// TIA Portal V17 export
// export: Created 2024-09-02T12:50:00.9082389Z, ExportSetting WithDefaults, DisplayName Totally Integrated Automation Portal, DisplayVersion V17, DisplayName TIA Portal Openness, DisplayVersion V17, DisplayName TIA Portal Version Control Interface, DisplayVersion V17, DisplayName STEP 7 Professional, DisplayVersion V17, DisplayName STEP 7 Safety, DisplayVersion V17, DisplayName WinCC Professional, DisplayVersion V17
FUNCTION_BLOCK "GraFB_Hand_41_50"   // FB1174, GRAPH
TITLE = GRAPH FB
AUTHOR : OlegFuehrus
FAMILY : SK
NAME : SK
VERSION : 0.1
// Hand functions / Handfunktionen
// stored: AcknowledgeErrorsRequired true, AutoNumber true, ExtensionBlockName LTLL_ManualGraphExt, GraphVersion 4.0, InitialValuesAcquisition false, IsIECCheckEnabled false, LanguageInNetworks LAD, LockOperatingMode false, PermanentILProcessingInMANMode true, SetENOAutomatically false, SkipSteps false, UDAEnableTagReadback false, WithAlarmHandling true
   // inherited from GRAPH_BASE
   VAR
      OFF_SQ_BASE : Bool;
   END_VAR
   VAR_INPUT
      OFF_SQ : Bool;
      INIT_SQ : Bool;
      ACK_EF : Bool;
      S_PREV : Bool;
      S_NEXT : Bool;
      SW_AUTO : Bool;
      SW_TAP : Bool;
      SW_MAN : Bool;
      S_SEL : Int;
      S_ON : Bool;
      S_OFF : Bool;
      T_PUSH : Bool;
   END_VAR
   VAR_OUTPUT
      S_NO : Int;
      S_MORE : Bool;
      S_ACTIVE : Bool;
      ERR_FLT : Bool;
      AUTO_ON : Bool;
      TAP_ON : Bool;
      MAN_ON : Bool;
   END_VAR
   VAR
      extBlock { S7_SetPoint := 'True'} : "LTLL_ManualGraphExt";
   END_VAR
   VAR_TEMP
      t_FrgHand : Bool;   // Freigabe Handbetrieb / Enable manual operation
      t_Service : Bool;   // Servicebetrieb aktiv / Service operation active
   END_VAR
BEGIN
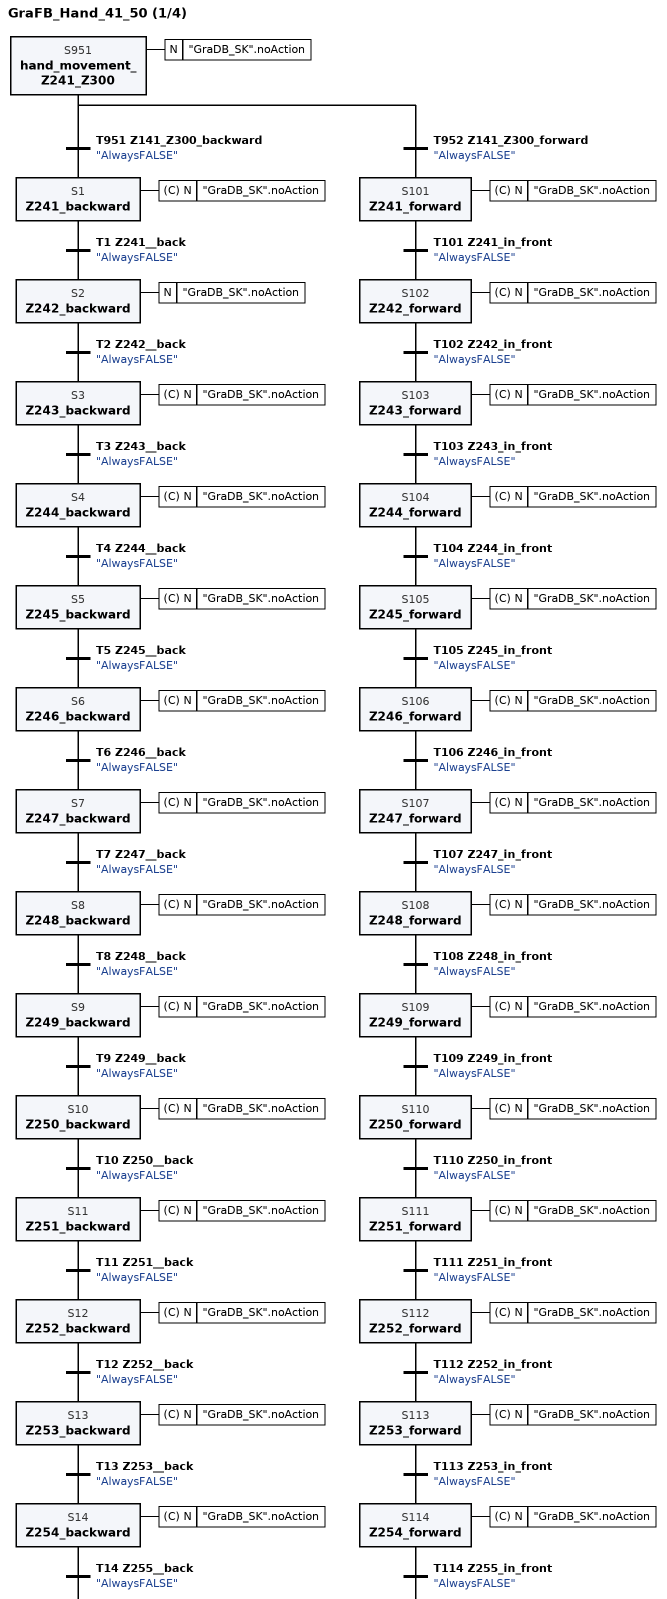
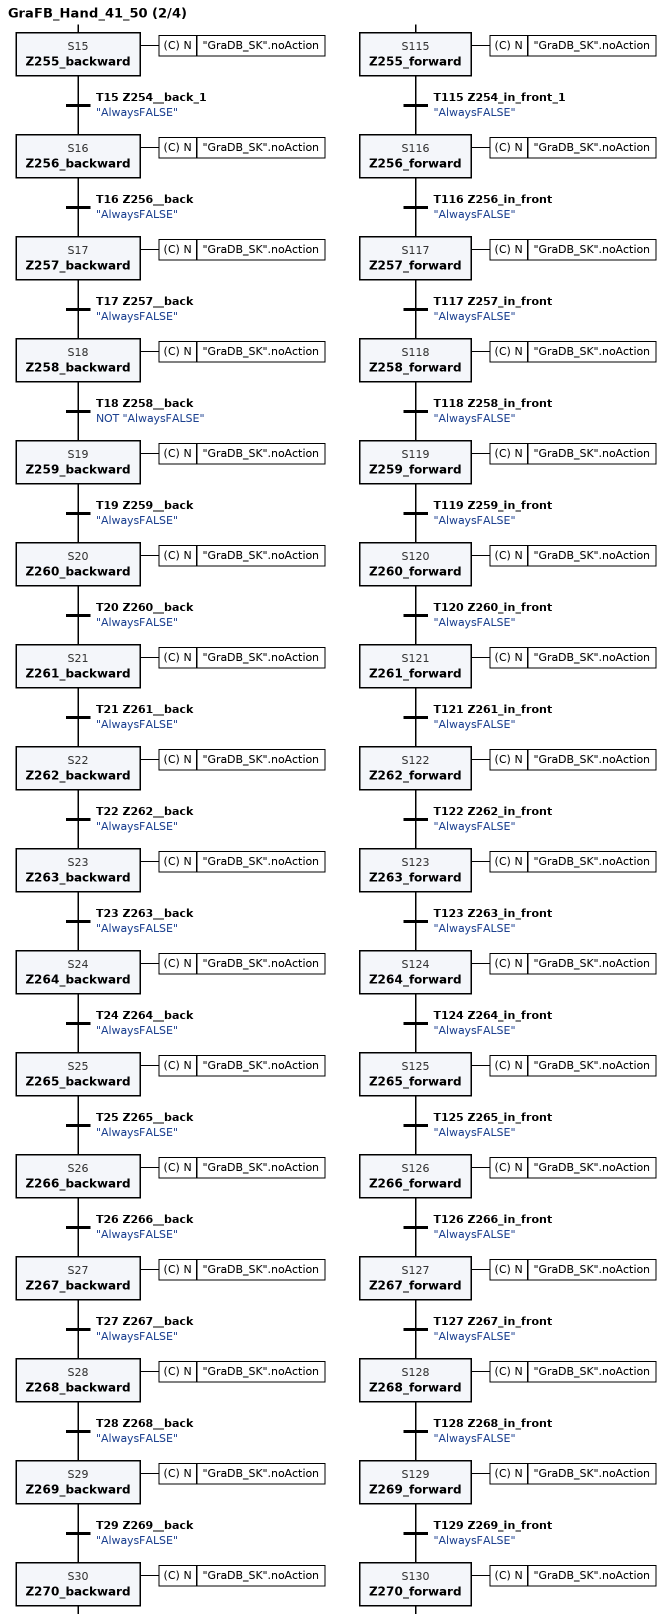
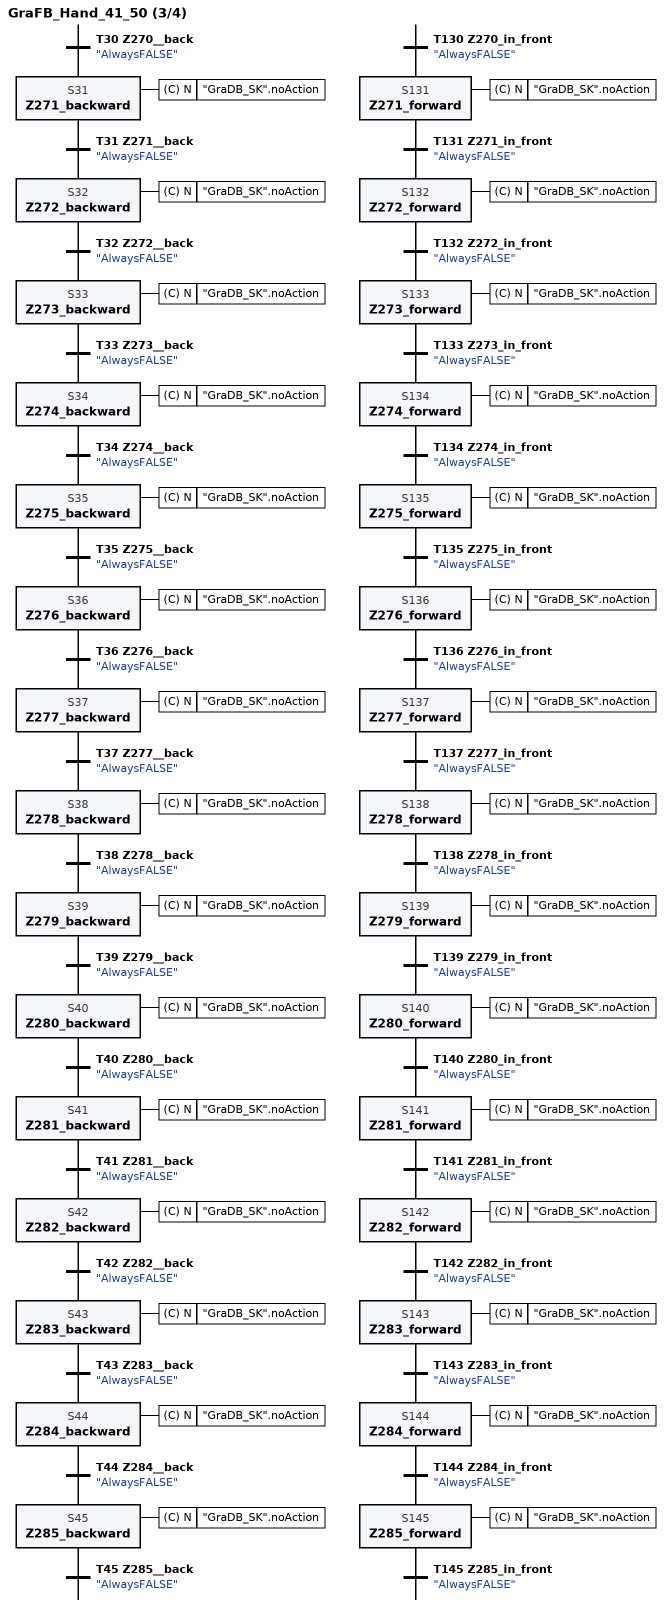
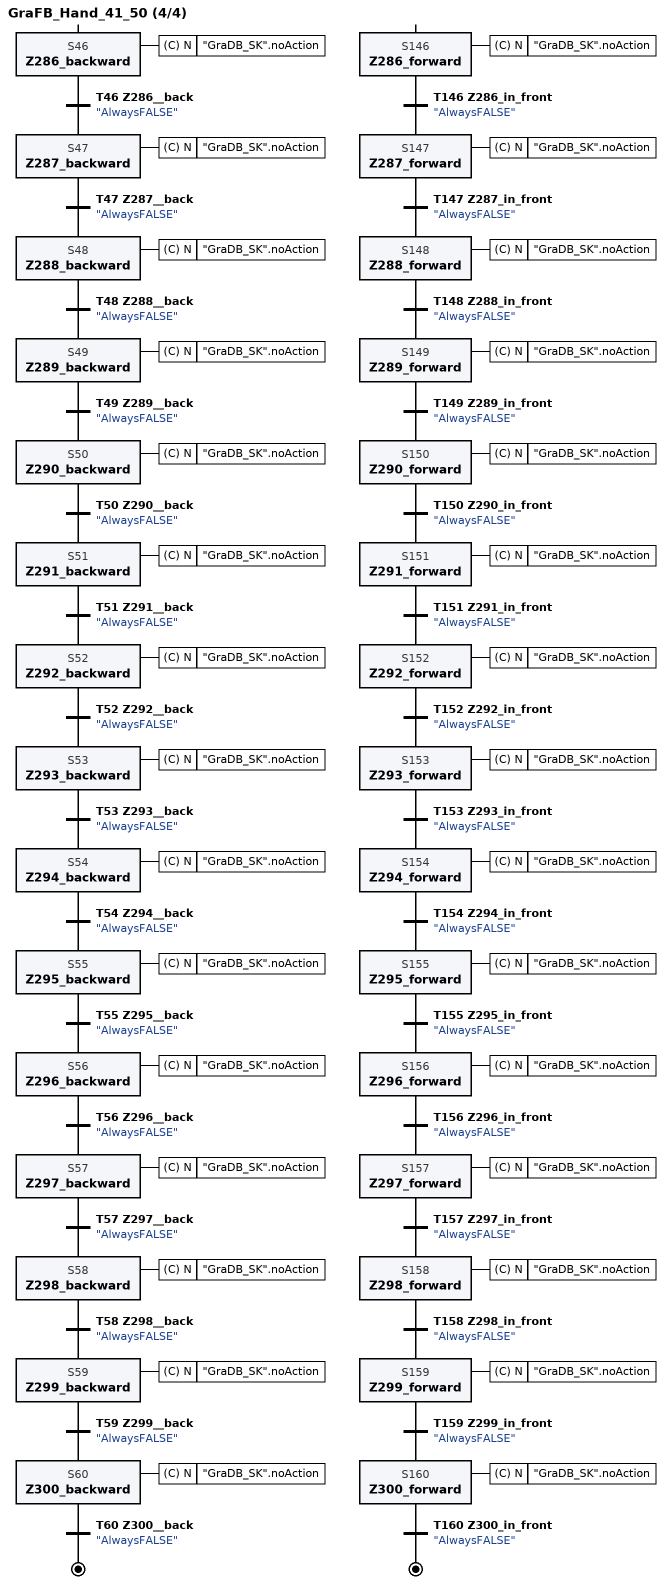
   // permanent pre-instructions
   NETWORK 1
   TITLE = HMI Lite Pass on data / HMI Lite Daten weiterreichen
      #extBlock.input := "LTLL_ManualGraphControl_OP70".screen[0].input;
   NETWORK 2
   TITLE = Instance DB Name query and pass on / Instanz DB Name abfragen und weiterreichen
      GetInstanceName(size := 0, OUT => #extBlock.input.instanceName);
   NETWORK 3
   TITLE = Interlocks Permanent machining, manual Approve and service / Interlocks Permanent Bearbeiten, Handfreigabe und Service
      IF NOT #RT_DATA.MOP.IL_PERM THEN #RT_DATA.MOP.IL_PERM := TRUE; END_IF;
      #t_FrgHand := "AnwDB_OperatingModes_OP70".BA[0]."mode_hand+start";
      #t_Service := "AnwDB_OperatingModes_OP70".BA[0].mode_service;

   // sequencer 1: Sequencer 1
   STEP hand_movement_Z241_Z300:   // S951, max time T#10S, warning time T#7S: Step commentary / Schrittkommentar
      interlock C := (none);   // hand_bereich_Z001_Z005
      supervision V := (none);   // hand_bereich_Z001_Z005
              N    "GraDB_SK".noAction
   END_STEP
   TRANSITION Z141_Z300_backward FROM hand_movement_Z241_Z300 TO Z241_backward   // T951
      := "AlwaysFALSE";
   END_TRANSITION
   TRANSITION Z141_Z300_forward FROM hand_movement_Z241_Z300 TO Z241_forward   // T952
      := "AlwaysFALSE";
   END_TRANSITION
   STEP Z241_backward:   // S1, max time T#10S, warning time T#7S
      interlock C := "AlwaysFALSE";   // Z241_zur
      supervision V := NOT #Z241__back.TT AND (#Z241_backward.T > T#5S);   // Z241_zur
      (C)     N    "GraDB_SK".noAction
   END_STEP
   TRANSITION Z241__back FROM Z241_backward TO Z242_backward   // T1
      := "AlwaysFALSE";
   END_TRANSITION
   STEP Z242_backward:   // S2, max time T#10S, warning time T#7S
      interlock C := "AlwaysFALSE";   // Z242_zur
      supervision V := NOT #Z242__back.TT AND (#Z242_backward.T > T#5S);   // Z242_zur
              N    "GraDB_SK".noAction
   END_STEP
   TRANSITION Z242__back FROM Z242_backward TO Z243_backward   // T2
      := "AlwaysFALSE";
   END_TRANSITION
   STEP Z243_backward:   // S3, max time T#10S, warning time T#7S
      interlock C := "AlwaysFALSE";   // Z243_zur
      supervision V := NOT #Z243__back.TT AND (#Z243_backward.T > T#5S);   // Z243_zur
      (C)     N    "GraDB_SK".noAction
   END_STEP
   TRANSITION Z243__back FROM Z243_backward TO Z244_backward   // T3
      := "AlwaysFALSE";
   END_TRANSITION
   STEP Z244_backward:   // S4, max time T#10S, warning time T#7S
      interlock C := "AlwaysFALSE";   // Z244_zur
      supervision V := NOT #Z244__back.TT AND (#Z244_backward.T > T#5S);   // Z244_zur
      (C)     N    "GraDB_SK".noAction
   END_STEP
   TRANSITION Z244__back FROM Z244_backward TO Z245_backward   // T4
      := "AlwaysFALSE";
   END_TRANSITION
   STEP Z245_backward:   // S5, max time T#10S, warning time T#7S
      interlock C := "AlwaysFALSE";   // Z245_zur
      supervision V := NOT #Z245__back.TT AND (#Z245_backward.T > T#5S);   // Z245_zur
      (C)     N    "GraDB_SK".noAction
   END_STEP
   TRANSITION Z245__back FROM Z245_backward TO Z246_backward   // T5
      := "AlwaysFALSE";
   END_TRANSITION
   STEP Z241_forward:   // S101, max time T#10S, warning time T#7S
      interlock C := "AlwaysFALSE";   // Z241_vor
      supervision V := NOT #Z241_in_front.TT AND (#Z241_forward.T > T#5S);   // Z241_vor
      (C)     N    "GraDB_SK".noAction
   END_STEP
   TRANSITION Z241_in_front FROM Z241_forward TO Z242_forward   // T101
      := "AlwaysFALSE";
   END_TRANSITION
   STEP Z242_forward:   // S102, max time T#10S, warning time T#7S
      interlock C := "AlwaysFALSE";   // Z242_vor
      supervision V := NOT #Z242_in_front.TT AND (#Z242_forward.T > T#5S);   // Z242_vor
      (C)     N    "GraDB_SK".noAction
   END_STEP
   TRANSITION Z242_in_front FROM Z242_forward TO Z243_forward   // T102
      := "AlwaysFALSE";
   END_TRANSITION
   STEP Z243_forward:   // S103, max time T#10S, warning time T#7S
      interlock C := "AlwaysFALSE";   // Z243_vor
      supervision V := NOT #Z243_in_front.TT AND (#Z243_forward.T > T#5S);   // Z243_vor
      (C)     N    "GraDB_SK".noAction
   END_STEP
   TRANSITION Z243_in_front FROM Z243_forward TO Z244_forward   // T103
      := "AlwaysFALSE";
   END_TRANSITION
   STEP Z244_forward:   // S104, max time T#10S, warning time T#7S
      interlock C := "AlwaysFALSE";   // Z244_vor
      supervision V := NOT #Z244_in_front.TT AND (#Z244_forward.T > T#5S);   // Z244_vor
      (C)     N    "GraDB_SK".noAction
   END_STEP
   TRANSITION Z244_in_front FROM Z244_forward TO Z245_forward   // T104
      := "AlwaysFALSE";
   END_TRANSITION
   STEP Z245_forward:   // S105, max time T#10S, warning time T#7S
      interlock C := "AlwaysFALSE";   // Z245_vor
      supervision V := NOT #Z245_in_front.TT AND (#Z245_forward.T > T#20S);   // Z245_vor
      (C)     N    "GraDB_SK".noAction
   END_STEP
   TRANSITION Z245_in_front FROM Z245_forward TO Z246_forward   // T105
      := "AlwaysFALSE";
   END_TRANSITION
   STEP Z246_backward:   // S6, max time T#10S, warning time T#7S: Cross transport 2 / Quertransport 2
      interlock C := "AlwaysFALSE";   // Z246_zur
      supervision V := NOT #Z246__back.TT AND (#Z246_backward.T > T#5S);   // Z246_zur
      (C)     N    "GraDB_SK".noAction
   END_STEP
   TRANSITION Z246__back FROM Z246_backward TO Z247_backward   // T6
      := "AlwaysFALSE";
   END_TRANSITION
   STEP Z247_backward:   // S7, max time T#10S, warning time T#7S
      interlock C := "AlwaysFALSE";   // Z247_zur
      supervision V := NOT #Z247__back.TT AND (#Z247_backward.T > T#5S);   // Z247_zur
      (C)     N    "GraDB_SK".noAction
   END_STEP
   TRANSITION Z247__back FROM Z247_backward TO Z248_backward   // T7
      := "AlwaysFALSE";
   END_TRANSITION
   STEP Z248_backward:   // S8, max time T#10S, warning time T#7S
      interlock C := "AlwaysFALSE";   // Z248_zur
      supervision V := NOT #Z248__back.TT AND (#Z248_backward.T > T#5S);   // Z248_zur
      (C)     N    "GraDB_SK".noAction
   END_STEP
   TRANSITION Z248__back FROM Z248_backward TO Z249_backward   // T8
      := "AlwaysFALSE";
   END_TRANSITION
   STEP Z249_backward:   // S9, max time T#10S, warning time T#7S
      interlock C := "AlwaysFALSE";   // Z249_zur
      supervision V := NOT #Z249__back.TT AND (#Z249_backward.T > T#5S);   // Z249_zur
      (C)     N    "GraDB_SK".noAction
   END_STEP
   TRANSITION Z249__back FROM Z249_backward TO Z250_backward   // T9
      := "AlwaysFALSE";
   END_TRANSITION
   STEP Z250_backward:   // S10, max time T#10S, warning time T#7S
      interlock C := "AlwaysFALSE";   // Z250_zur
      supervision V := NOT #Z250__back.TT AND (#Z250_backward.T > T#5S);   // Z250_zur
      (C)     N    "GraDB_SK".noAction
   END_STEP
   TRANSITION Z250__back FROM Z250_backward TO Z251_backward   // T10
      := "AlwaysFALSE";
   END_TRANSITION
   STEP Z246_forward:   // S106, max time T#10S, warning time T#7S
      interlock C := "AlwaysFALSE";   // Z246_vor
      supervision V := NOT #Z246_in_front.TT AND (#Z246_forward.T > T#5S);   // Z246_vor
      (C)     N    "GraDB_SK".noAction
   END_STEP
   TRANSITION Z246_in_front FROM Z246_forward TO Z247_forward   // T106
      := "AlwaysFALSE";
   END_TRANSITION
   STEP Z247_forward:   // S107, max time T#10S, warning time T#7S
      interlock C := "AlwaysFALSE";   // Z247_vor
      supervision V := NOT #Z247_in_front.TT AND (#Z247_forward.T > T#5S);   // Z247_vor
      (C)     N    "GraDB_SK".noAction
   END_STEP
   TRANSITION Z247_in_front FROM Z247_forward TO Z248_forward   // T107
      := "AlwaysFALSE";
   END_TRANSITION
   STEP Z248_forward:   // S108, max time T#10S, warning time T#7S
      interlock C := "AlwaysFALSE";   // Z248_vor
      supervision V := NOT #Z248_in_front.TT AND (#Z248_forward.T > T#5S);   // Z248_vor
      (C)     N    "GraDB_SK".noAction
   END_STEP
   TRANSITION Z248_in_front FROM Z248_forward TO Z249_forward   // T108
      := "AlwaysFALSE";
   END_TRANSITION
   STEP Z249_forward:   // S109, max time T#10S, warning time T#7S
      interlock C := "AlwaysFALSE";   // Z249_vor
      supervision V := NOT #Z249_in_front.TT AND (#Z249_forward.T > T#5S);   // Z249_vor
      (C)     N    "GraDB_SK".noAction
   END_STEP
   TRANSITION Z249_in_front FROM Z249_forward TO Z250_forward   // T109
      := "AlwaysFALSE";
   END_TRANSITION
   STEP Z250_forward:   // S110, max time T#10S, warning time T#7S
      interlock C := "AlwaysFALSE";   // Z250_vor
      supervision V := NOT #Z250_in_front.TT AND (#Z250_forward.T > T#5S);   // Z250_vor
      (C)     N    "GraDB_SK".noAction
   END_STEP
   TRANSITION Z250_in_front FROM Z250_forward TO Z251_forward   // T110
      := "AlwaysFALSE";
   END_TRANSITION
   STEP Z251_backward:   // S11, max time T#10S, warning time T#7S
      interlock C := "AlwaysFALSE";   // Z251_zur
      supervision V := NOT #Z251__back.TT AND (#Z251_backward.T > T#5S);   // Z251_zur
      (C)     N    "GraDB_SK".noAction
   END_STEP
   TRANSITION Z251__back FROM Z251_backward TO Z252_backward   // T11
      := "AlwaysFALSE";
   END_TRANSITION
   STEP Z252_backward:   // S12, max time T#10S, warning time T#7S
      interlock C := "AlwaysFALSE";   // Z252_zur
      supervision V := NOT #Z252__back.TT AND (#Z252_backward.T > T#5S);   // Z252_zur
      (C)     N    "GraDB_SK".noAction
   END_STEP
   TRANSITION Z252__back FROM Z252_backward TO Z253_backward   // T12
      := "AlwaysFALSE";
   END_TRANSITION
   STEP Z253_backward:   // S13, max time T#10S, warning time T#7S
      interlock C := "AlwaysFALSE";   // Z253_zur
      supervision V := NOT #Z253__back.TT AND (#Z253_backward.T > T#5S);   // Z253_zur
      (C)     N    "GraDB_SK".noAction
   END_STEP
   TRANSITION Z253__back FROM Z253_backward TO Z254_backward   // T13
      := "AlwaysFALSE";
   END_TRANSITION
   STEP Z254_backward:   // S14, max time T#10S, warning time T#7S
      interlock C := "AlwaysFALSE";   // Z255_zur
      supervision V := NOT #Z255__back.TT AND (#Z254_backward.T > T#5S);   // Z255_zur
      (C)     N    "GraDB_SK".noAction
   END_STEP
   TRANSITION Z255__back FROM Z254_backward TO Z255_backward   // T14
      := "AlwaysFALSE";
   END_TRANSITION
   STEP Z255_backward:   // S15, max time T#10S, warning time T#7S
      interlock C := "AlwaysFALSE";   // Z254_zur
      supervision V := NOT #Z256__back.TT AND (#Z255_backward.T > T#5S);   // Z25_zur
      (C)     N    "GraDB_SK".noAction
   END_STEP
   TRANSITION Z254__back_1 FROM Z255_backward TO Z256_backward   // T15
      := "AlwaysFALSE";
   END_TRANSITION
   STEP Z251_forward:   // S111, max time T#10S, warning time T#7S
      interlock C := "AlwaysFALSE";   // Z251_vor
      supervision V := NOT #Z251_in_front.TT AND (#Z251_forward.T > T#5S);   // Z251_vor
      (C)     N    "GraDB_SK".noAction
   END_STEP
   TRANSITION Z251_in_front FROM Z251_forward TO Z252_forward   // T111
      := "AlwaysFALSE";
   END_TRANSITION
   STEP Z252_forward:   // S112, max time T#10S, warning time T#7S
      interlock C := "AlwaysFALSE";   // Z252_vor
      supervision V := NOT #Z252_in_front.TT AND (#Z252_forward.T > T#5S);   // Z252_vor
      (C)     N    "GraDB_SK".noAction
   END_STEP
   TRANSITION Z252_in_front FROM Z252_forward TO Z253_forward   // T112
      := "AlwaysFALSE";
   END_TRANSITION
   STEP Z253_forward:   // S113, max time T#10S, warning time T#7S
      interlock C := "AlwaysFALSE";   // Z253_vor
      supervision V := NOT #Z253_in_front.TT AND (#Z253_forward.T > T#5S);   // Z253_vor
      (C)     N    "GraDB_SK".noAction
   END_STEP
   TRANSITION Z253_in_front FROM Z253_forward TO Z254_forward   // T113
      := "AlwaysFALSE";
   END_TRANSITION
   STEP Z254_forward:   // S114, max time T#10S, warning time T#7S
      interlock C := "AlwaysFALSE";   // Z255_vor
      supervision V := NOT #Z255_in_front.TT AND (#Z254_forward.T > T#5S);   // Z255_vor
      (C)     N    "GraDB_SK".noAction
   END_STEP
   TRANSITION Z255_in_front FROM Z254_forward TO Z255_forward   // T114
      := "AlwaysFALSE";
   END_TRANSITION
   STEP Z255_forward:   // S115, max time T#10S, warning time T#7S
      interlock C := "AlwaysFALSE";   // Z254_vor
      supervision V := NOT #Z256_in_front.TT AND (#Z255_forward.T > T#5S);   // Z254_vor
      (C)     N    "GraDB_SK".noAction
   END_STEP
   TRANSITION Z254_in_front_1 FROM Z255_forward TO Z256_forward   // T115
      := "AlwaysFALSE";
   END_TRANSITION
   STEP Z256_backward:   // S16, max time T#10S, warning time T#7S
      interlock C := "AlwaysFALSE";   // Z256_zur
      supervision V := NOT #Z256__back.TT AND (#Z256_backward.T > T#5S);   // Z256_zur
      (C)     N    "GraDB_SK".noAction
   END_STEP
   TRANSITION Z256__back FROM Z256_backward TO Z257_backward   // T16
      := "AlwaysFALSE";
   END_TRANSITION
   STEP Z257_backward:   // S17, max time T#10S, warning time T#7S
      interlock C := "AlwaysFALSE";   // Z257_zur
      supervision V := NOT #Z257__back.TT AND (#Z257_backward.T > T#5S);   // Z257_zur
      (C)     N    "GraDB_SK".noAction
   END_STEP
   TRANSITION Z257__back FROM Z257_backward TO Z258_backward   // T17
      := "AlwaysFALSE";
   END_TRANSITION
   STEP Z258_backward:   // S18, max time T#10S, warning time T#7S
      interlock C := "AlwaysFALSE";   // Z258_zur
      supervision V := NOT #Z258__back.TT AND (#Z258_backward.T > T#5S);   // Z258_zur
      (C)     N    "GraDB_SK".noAction
   END_STEP
   TRANSITION Z258__back FROM Z258_backward TO Z259_backward   // T18
      := NOT "AlwaysFALSE";
   END_TRANSITION
   STEP Z259_backward:   // S19, max time T#10S, warning time T#7S
      interlock C := "AlwaysFALSE";   // Z259_zur
      supervision V := NOT #Z259__back.TT AND (#Z259_backward.T > T#5S);   // Z259_zur
      (C)     N    "GraDB_SK".noAction
   END_STEP
   TRANSITION Z259__back FROM Z259_backward TO Z260_backward   // T19
      := "AlwaysFALSE";
   END_TRANSITION
   STEP Z260_backward:   // S20, max time T#10S, warning time T#7S
      interlock C := "AlwaysFALSE";   // Z260_zur
      supervision V := NOT #Z260__back.TT AND (#Z260_backward.T > T#5S);   // Z260_zur
      (C)     N    "GraDB_SK".noAction
   END_STEP
   TRANSITION Z260__back FROM Z260_backward TO Z261_backward   // T20
      := "AlwaysFALSE";
   END_TRANSITION
   STEP Z256_forward:   // S116, max time T#10S, warning time T#7S
      interlock C := "AlwaysFALSE";   // Z256_vor
      supervision V := NOT #Z256_in_front.TT AND (#Z256_forward.T > T#5S);   // Z256_vor
      (C)     N    "GraDB_SK".noAction
   END_STEP
   TRANSITION Z256_in_front FROM Z256_forward TO Z257_forward   // T116
      := "AlwaysFALSE";
   END_TRANSITION
   STEP Z257_forward:   // S117, max time T#10S, warning time T#7S
      interlock C := "AlwaysFALSE";   // Z257_vor
      supervision V := NOT #Z257_in_front.TT AND (#Z257_forward.T > T#5S);   // Z257_vor
      (C)     N    "GraDB_SK".noAction
   END_STEP
   TRANSITION Z257_in_front FROM Z257_forward TO Z258_forward   // T117
      := "AlwaysFALSE";
   END_TRANSITION
   STEP Z258_forward:   // S118, max time T#10S, warning time T#7S
      interlock C := "AlwaysFALSE";   // Z258_vor
      supervision V := NOT #Z258_in_front.TT AND (#Z258_forward.T > T#5S);   // Z258_vor
      (C)     N    "GraDB_SK".noAction
   END_STEP
   TRANSITION Z258_in_front FROM Z258_forward TO Z259_forward   // T118
      := "AlwaysFALSE";
   END_TRANSITION
   STEP Z259_forward:   // S119, max time T#10S, warning time T#7S
      interlock C := "AlwaysFALSE";   // Z259_vor
      supervision V := NOT #Z259_in_front.TT AND (#Z259_forward.T > T#5S);   // Z259_vor
      (C)     N    "GraDB_SK".noAction
   END_STEP
   TRANSITION Z259_in_front FROM Z259_forward TO Z260_forward   // T119
      := "AlwaysFALSE";
   END_TRANSITION
   STEP Z260_forward:   // S120, max time T#10S, warning time T#7S
      interlock C := "AlwaysFALSE";   // Z260_vor
      supervision V := NOT #Z260_in_front.TT AND (#Z260_forward.T > T#5S);   // Z260_vor
      (C)     N    "GraDB_SK".noAction
   END_STEP
   TRANSITION Z260_in_front FROM Z260_forward TO Z261_forward   // T120
      := "AlwaysFALSE";
   END_TRANSITION
   STEP Z261_backward:   // S21, max time T#10S, warning time T#7S
      interlock C := "AlwaysFALSE";   // Z261_zur
      supervision V := NOT #Z261__back.TT AND (#Z261_backward.T > T#10S);   // Z261_zur
      (C)     N    "GraDB_SK".noAction
   END_STEP
   TRANSITION Z261__back FROM Z261_backward TO Z262_backward   // T21
      := "AlwaysFALSE";
   END_TRANSITION
   STEP Z262_backward:   // S22, max time T#10S, warning time T#7S
      interlock C := "AlwaysFALSE";   // Z262_zur
      supervision V := NOT #Z262__back.TT AND (#Z262_backward.T > T#10S);   // Z262_zur
      (C)     N    "GraDB_SK".noAction
   END_STEP
   TRANSITION Z262__back FROM Z262_backward TO Z263_backward   // T22
      := "AlwaysFALSE";
   END_TRANSITION
   STEP Z263_backward:   // S23, max time T#10S, warning time T#7S
      interlock C := "AlwaysFALSE";   // Z263_zur
      supervision V := NOT #Z263__back.TT AND (#Z263_backward.T > T#10S);   // Z263_zur
      (C)     N    "GraDB_SK".noAction
   END_STEP
   TRANSITION Z263__back FROM Z263_backward TO Z264_backward   // T23
      := "AlwaysFALSE";
   END_TRANSITION
   STEP Z264_backward:   // S24, max time T#10S, warning time T#7S
      interlock C := "AlwaysFALSE";   // Z264_zur
      supervision V := NOT #Z264__back.TT AND (#Z264_backward.T > T#5S);   // Z264_zur
      (C)     N    "GraDB_SK".noAction
   END_STEP
   TRANSITION Z264__back FROM Z264_backward TO Z265_backward   // T24
      := "AlwaysFALSE";
   END_TRANSITION
   STEP Z265_backward:   // S25, max time T#10S, warning time T#7S
      interlock C := "AlwaysFALSE";   // Z265_zur
      supervision V := NOT #Z265__back.TT AND (#Z265_backward.T > T#5S);   // Z265_zur
      (C)     N    "GraDB_SK".noAction
   END_STEP
   TRANSITION Z265__back FROM Z265_backward TO Z266_backward   // T25
      := "AlwaysFALSE";
   END_TRANSITION
   STEP Z261_forward:   // S121, max time T#10S, warning time T#7S
      interlock C := "AlwaysFALSE";   // Z261_vor
      supervision V := NOT #Z261_in_front.TT AND (#Z261_forward.T > T#5S);   // Z261_vor
      (C)     N    "GraDB_SK".noAction
   END_STEP
   TRANSITION Z261_in_front FROM Z261_forward TO Z262_forward   // T121
      := "AlwaysFALSE";
   END_TRANSITION
   STEP Z262_forward:   // S122, max time T#10S, warning time T#7S
      interlock C := "AlwaysFALSE";   // Z262_vor
      supervision V := NOT #Z262_in_front.TT AND (#Z262_forward.T > T#10S);   // Z262_vor
      (C)     N    "GraDB_SK".noAction
   END_STEP
   TRANSITION Z262_in_front FROM Z262_forward TO Z263_forward   // T122
      := "AlwaysFALSE";
   END_TRANSITION
   STEP Z263_forward:   // S123, max time T#10S, warning time T#7S
      interlock C := "AlwaysFALSE";   // Z263_vor
      supervision V := NOT #Z263_in_front.TT AND (#Z263_forward.T > T#10S);   // Z263_vor
      (C)     N    "GraDB_SK".noAction
   END_STEP
   TRANSITION Z263_in_front FROM Z263_forward TO Z264_forward   // T123
      := "AlwaysFALSE";
   END_TRANSITION
   STEP Z264_forward:   // S124, max time T#10S, warning time T#7S
      interlock C := "AlwaysFALSE";   // Z264_vor
      supervision V := NOT #Z264_in_front.TT AND (#Z264_forward.T > T#5S);   // Z264_vor
      (C)     N    "GraDB_SK".noAction
   END_STEP
   TRANSITION Z264_in_front FROM Z264_forward TO Z265_forward   // T124
      := "AlwaysFALSE";
   END_TRANSITION
   STEP Z265_forward:   // S125, max time T#10S, warning time T#7S
      interlock C := "AlwaysFALSE";   // Z265_vor
      supervision V := NOT #Z265_in_front.TT AND (#Z265_forward.T > T#5S);   // Z265_vor
      (C)     N    "GraDB_SK".noAction
   END_STEP
   TRANSITION Z265_in_front FROM Z265_forward TO Z266_forward   // T125
      := "AlwaysFALSE";
   END_TRANSITION
   STEP Z266_backward:   // S26, max time T#10S, warning time T#7S
      interlock C := "AlwaysFALSE";   // Z266_zur
      supervision V := NOT #Z266__back.TT AND (#Z266_backward.T > T#5S);   // Z266_zur
      (C)     N    "GraDB_SK".noAction
   END_STEP
   TRANSITION Z266__back FROM Z266_backward TO Z267_backward   // T26
      := "AlwaysFALSE";
   END_TRANSITION
   STEP Z267_backward:   // S27, max time T#10S, warning time T#7S
      interlock C := "AlwaysFALSE";   // Z267_zur
      supervision V := NOT #Z267__back.TT AND (#Z267_backward.T > T#5S);   // Z267_zur
      (C)     N    "GraDB_SK".noAction
   END_STEP
   TRANSITION Z267__back FROM Z267_backward TO Z268_backward   // T27
      := "AlwaysFALSE";
   END_TRANSITION
   STEP Z268_backward:   // S28, max time T#10S, warning time T#7S
      interlock C := "AlwaysFALSE";   // Z268_zur
      supervision V := NOT #Z268__back.TT AND (#Z268_backward.T > T#5S);   // Z268_zur
      (C)     N    "GraDB_SK".noAction
   END_STEP
   TRANSITION Z268__back FROM Z268_backward TO Z269_backward   // T28
      := "AlwaysFALSE";
   END_TRANSITION
   STEP Z269_backward:   // S29, max time T#10S, warning time T#7S
      interlock C := "AlwaysFALSE";   // Z269_zur
      supervision V := NOT #Z269__back.TT AND (#Z269_backward.T > T#5S);   // Z269_zur
      (C)     N    "GraDB_SK".noAction
   END_STEP
   TRANSITION Z269__back FROM Z269_backward TO Z270_backward   // T29
      := "AlwaysFALSE";
   END_TRANSITION
   STEP Z270_backward:   // S30, max time T#10S, warning time T#7S
      interlock C := "AlwaysFALSE";   // Z270_zur
      supervision V := NOT #Z270__back.TT AND (#Z270_backward.T > T#5S);   // Z270_zur
      (C)     N    "GraDB_SK".noAction
   END_STEP
   TRANSITION Z270__back FROM Z270_backward TO Z271_backward   // T30
      := "AlwaysFALSE";
   END_TRANSITION
   STEP Z266_forward:   // S126, max time T#10S, warning time T#7S
      interlock C := "AlwaysFALSE";   // Z266_vor
      supervision V := NOT #Z266_in_front.TT AND (#Z266_forward.T > T#5S);   // Z266_vor
      (C)     N    "GraDB_SK".noAction
   END_STEP
   TRANSITION Z266_in_front FROM Z266_forward TO Z267_forward   // T126
      := "AlwaysFALSE";
   END_TRANSITION
   STEP Z267_forward:   // S127, max time T#10S, warning time T#7S
      interlock C := "AlwaysFALSE";   // Z267_vor
      supervision V := NOT #Z267_in_front.TT AND (#Z267_forward.T > T#5S);   // Z267_vor
      (C)     N    "GraDB_SK".noAction
   END_STEP
   TRANSITION Z267_in_front FROM Z267_forward TO Z268_forward   // T127
      := "AlwaysFALSE";
   END_TRANSITION
   STEP Z268_forward:   // S128, max time T#10S, warning time T#7S
      interlock C := "AlwaysFALSE";   // Z268_vor
      supervision V := NOT #Z268_in_front.TT AND (#Z268_forward.T > T#5S);   // Z268_vor
      (C)     N    "GraDB_SK".noAction
   END_STEP
   TRANSITION Z268_in_front FROM Z268_forward TO Z269_forward   // T128
      := "AlwaysFALSE";
   END_TRANSITION
   STEP Z269_forward:   // S129, max time T#10S, warning time T#7S
      interlock C := "AlwaysFALSE";   // Z269_vor
      supervision V := NOT #Z269_in_front.TT AND (#Z269_forward.T > T#5S);   // Z269_vor
      (C)     N    "GraDB_SK".noAction
   END_STEP
   TRANSITION Z269_in_front FROM Z269_forward TO Z270_forward   // T129
      := "AlwaysFALSE";
   END_TRANSITION
   STEP Z270_forward:   // S130, max time T#10S, warning time T#7S
      interlock C := "AlwaysFALSE";   // Z270_vor
      supervision V := NOT #Z270_in_front.TT AND (#Z270_forward.T > T#5S);   // Z270_vor
      (C)     N    "GraDB_SK".noAction
   END_STEP
   TRANSITION Z270_in_front FROM Z270_forward TO Z271_forward   // T130
      := "AlwaysFALSE";
   END_TRANSITION
   STEP Z271_backward:   // S31, max time T#10S, warning time T#7S: Step commentary / Schrittkommentar
      interlock C := "AlwaysFALSE";   // Z271_zur
      supervision V := NOT #Z271__back.TT AND (#Z271_backward.T > T#5S);   // Z271_zur
      (C)     N    "GraDB_SK".noAction
   END_STEP
   TRANSITION Z271__back FROM Z271_backward TO Z272_backward   // T31
      := "AlwaysFALSE";
   END_TRANSITION
   STEP Z272_backward:   // S32, max time T#10S, warning time T#7S: Step commentary / Schrittkommentar
      interlock C := "AlwaysFALSE";   // Z272_zur
      supervision V := NOT #Z272__back.TT AND (#Z272_backward.T > T#5S);   // Z272_zur
      (C)     N    "GraDB_SK".noAction
   END_STEP
   TRANSITION Z272__back FROM Z272_backward TO Z273_backward   // T32
      := "AlwaysFALSE";
   END_TRANSITION
   STEP Z273_backward:   // S33, max time T#10S, warning time T#7S: Step commentary / Schrittkommentar
      interlock C := "AlwaysFALSE";   // Z273_zur
      supervision V := NOT #Z273__back.TT AND (#Z273_backward.T > T#5S);   // Z273_zur
      (C)     N    "GraDB_SK".noAction
   END_STEP
   TRANSITION Z273__back FROM Z273_backward TO Z274_backward   // T33
      := "AlwaysFALSE";
   END_TRANSITION
   STEP Z274_backward:   // S34, max time T#10S, warning time T#7S: Step commentary / Schrittkommentar
      interlock C := "AlwaysFALSE";   // Z274_zur
      supervision V := NOT #Z274__back.TT AND (#Z274_backward.T > T#5S);   // Z274_zur
      (C)     N    "GraDB_SK".noAction
   END_STEP
   TRANSITION Z274__back FROM Z274_backward TO Z275_backward   // T34
      := "AlwaysFALSE";
   END_TRANSITION
   STEP Z275_backward:   // S35, max time T#10S, warning time T#7S: Step commentary / Schrittkommentar
      interlock C := "AlwaysFALSE";   // Z275_zur
      supervision V := NOT #Z275__back.TT AND (#Z275_backward.T > T#5S);   // Z275_zur
      (C)     N    "GraDB_SK".noAction
   END_STEP
   TRANSITION Z275__back FROM Z275_backward TO Z276_backward   // T35
      := "AlwaysFALSE";
   END_TRANSITION
   STEP Z271_forward:   // S131, max time T#10S, warning time T#7S: Step commentary / Schrittkommentar
      interlock C := "AlwaysFALSE";   // Z271_vor
      supervision V := NOT #Z271_in_front.TT AND (#Z271_forward.T > T#5S);   // Z271_vor
      (C)     N    "GraDB_SK".noAction
   END_STEP
   TRANSITION Z271_in_front FROM Z271_forward TO Z272_forward   // T131
      := "AlwaysFALSE";
   END_TRANSITION
   STEP Z272_forward:   // S132, max time T#10S, warning time T#7S: Step commentary / Schrittkommentar
      interlock C := "AlwaysFALSE";   // Z272_vor
      supervision V := NOT #Z272_in_front.TT AND (#Z272_forward.T > T#5S);   // Z272_vor
      (C)     N    "GraDB_SK".noAction
   END_STEP
   TRANSITION Z272_in_front FROM Z272_forward TO Z273_forward   // T132
      := "AlwaysFALSE";
   END_TRANSITION
   STEP Z273_forward:   // S133, max time T#10S, warning time T#7S: Step commentary / Schrittkommentar
      interlock C := "AlwaysFALSE";   // Z273_vor
      supervision V := NOT #Z273_in_front.TT AND (#Z273_forward.T > T#5S);   // Z273_vor
      (C)     N    "GraDB_SK".noAction
   END_STEP
   TRANSITION Z273_in_front FROM Z273_forward TO Z274_forward   // T133
      := "AlwaysFALSE";
   END_TRANSITION
   STEP Z274_forward:   // S134, max time T#10S, warning time T#7S: Step commentary / Schrittkommentar
      interlock C := "AlwaysFALSE";   // Z274_vor
      supervision V := NOT #Z274_in_front.TT AND (#Z274_forward.T > T#5S);   // Z274_vor
      (C)     N    "GraDB_SK".noAction
   END_STEP
   TRANSITION Z274_in_front FROM Z274_forward TO Z275_forward   // T134
      := "AlwaysFALSE";
   END_TRANSITION
   STEP Z275_forward:   // S135, max time T#10S, warning time T#7S: Step commentary / Schrittkommentar
      interlock C := "AlwaysFALSE";   // Z275_vor
      supervision V := NOT #Z275_in_front.TT AND (#Z275_forward.T > T#5S);   // Z275_vor
      (C)     N    "GraDB_SK".noAction
   END_STEP
   TRANSITION Z275_in_front FROM Z275_forward TO Z276_forward   // T135
      := "AlwaysFALSE";
   END_TRANSITION
   STEP Z276_backward:   // S36, max time T#10S, warning time T#7S: Step commentary / Schrittkommentar
      interlock C := "AlwaysFALSE";   // Z276_zur
      supervision V := NOT #Z276__back.TT AND (#Z276_backward.T > T#5S);   // Z276_zur
      (C)     N    "GraDB_SK".noAction
   END_STEP
   TRANSITION Z276__back FROM Z276_backward TO Z277_backward   // T36
      := "AlwaysFALSE";
   END_TRANSITION
   STEP Z277_backward:   // S37, max time T#10S, warning time T#7S: Step commentary / Schrittkommentar
      interlock C := "AlwaysFALSE";   // Z277_zur
      supervision V := NOT #Z277__back.TT AND (#Z277_backward.T > T#5S);   // Z277_zur
      (C)     N    "GraDB_SK".noAction
   END_STEP
   TRANSITION Z277__back FROM Z277_backward TO Z278_backward   // T37
      := "AlwaysFALSE";
   END_TRANSITION
   STEP Z278_backward:   // S38, max time T#10S, warning time T#7S: Step commentary / Schrittkommentar
      interlock C := "AlwaysFALSE";   // Z278_zur
      supervision V := NOT #Z278__back.TT AND (#Z278_backward.T > T#5S);   // Z278_zur
      (C)     N    "GraDB_SK".noAction
   END_STEP
   TRANSITION Z278__back FROM Z278_backward TO Z279_backward   // T38
      := "AlwaysFALSE";
   END_TRANSITION
   STEP Z279_backward:   // S39, max time T#10S, warning time T#7S: Step commentary / Schrittkommentar
      interlock C := "AlwaysFALSE";   // Z279_zur
      supervision V := NOT #Z279__back.TT AND (#Z279_backward.T > T#5S);   // Z279_zur
      (C)     N    "GraDB_SK".noAction
   END_STEP
   TRANSITION Z279__back FROM Z279_backward TO Z280_backward   // T39
      := "AlwaysFALSE";
   END_TRANSITION
   STEP Z280_backward:   // S40, max time T#10S, warning time T#7S: Step commentary / Schrittkommentar
      interlock C := "AlwaysFALSE";   // Z280_zur
      supervision V := NOT #Z280__back.TT AND (#Z280_backward.T > T#5S);   // Z280_zur
      (C)     N    "GraDB_SK".noAction
   END_STEP
   TRANSITION Z280__back FROM Z280_backward TO Z281_backward   // T40
      := "AlwaysFALSE";
   END_TRANSITION
   STEP Z276_forward:   // S136, max time T#10S, warning time T#7S: Step commentary / Schrittkommentar
      interlock C := "AlwaysFALSE";   // Z276_vor
      supervision V := NOT #Z276_in_front.TT AND (#Z276_forward.T > T#5S);   // Z276_vor
      (C)     N    "GraDB_SK".noAction
   END_STEP
   TRANSITION Z276_in_front FROM Z276_forward TO Z277_forward   // T136
      := "AlwaysFALSE";
   END_TRANSITION
   STEP Z277_forward:   // S137, max time T#10S, warning time T#7S: Step commentary / Schrittkommentar
      interlock C := "AlwaysFALSE";   // Z277_vor
      supervision V := NOT #Z277_in_front.TT AND (#Z277_forward.T > T#5S);   // Z277_vor
      (C)     N    "GraDB_SK".noAction
   END_STEP
   TRANSITION Z277_in_front FROM Z277_forward TO Z278_forward   // T137
      := "AlwaysFALSE";
   END_TRANSITION
   STEP Z278_forward:   // S138, max time T#10S, warning time T#7S: Step commentary / Schrittkommentar
      interlock C := "AlwaysFALSE";   // Z278_vor
      supervision V := NOT #Z278_in_front.TT AND (#Z278_forward.T > T#5S);   // Z278_vor
      (C)     N    "GraDB_SK".noAction
   END_STEP
   TRANSITION Z278_in_front FROM Z278_forward TO Z279_forward   // T138
      := "AlwaysFALSE";
   END_TRANSITION
   STEP Z279_forward:   // S139, max time T#10S, warning time T#7S: Step commentary / Schrittkommentar
      interlock C := "AlwaysFALSE";   // Z279_vor
      supervision V := NOT #Z279_in_front.TT AND (#Z279_forward.T > T#5S);   // Z279_vor
      (C)     N    "GraDB_SK".noAction
   END_STEP
   TRANSITION Z279_in_front FROM Z279_forward TO Z280_forward   // T139
      := "AlwaysFALSE";
   END_TRANSITION
   STEP Z280_forward:   // S140, max time T#10S, warning time T#7S: Step commentary / Schrittkommentar
      interlock C := "AlwaysFALSE";   // Z280_vor
      supervision V := NOT #Z280_in_front.TT AND (#Z280_forward.T > T#5S);   // Z280_vor
      (C)     N    "GraDB_SK".noAction
   END_STEP
   TRANSITION Z280_in_front FROM Z280_forward TO Z281_forward   // T140
      := "AlwaysFALSE";
   END_TRANSITION
   STEP Z281_backward:   // S41, max time T#10S, warning time T#7S: Step commentary / Schrittkommentar
      interlock C := "AlwaysFALSE";   // Z281_zur
      supervision V := NOT #Z281__back.TT AND (#Z281_backward.T > T#5S);   // Z281_zur
      (C)     N    "GraDB_SK".noAction
   END_STEP
   TRANSITION Z281__back FROM Z281_backward TO Z282_backward   // T41
      := "AlwaysFALSE";
   END_TRANSITION
   STEP Z282_backward:   // S42, max time T#10S, warning time T#7S: Step commentary / Schrittkommentar
      interlock C := "AlwaysFALSE";   // Z282_zur
      supervision V := NOT #Z282__back.TT AND (#Z282_backward.T > T#5S);   // Z282_zur
      (C)     N    "GraDB_SK".noAction
   END_STEP
   TRANSITION Z282__back FROM Z282_backward TO Z283_backward   // T42
      := "AlwaysFALSE";
   END_TRANSITION
   STEP Z283_backward:   // S43, max time T#10S, warning time T#7S: Step commentary / Schrittkommentar
      interlock C := "AlwaysFALSE";   // Z283_zur
      supervision V := NOT #Z283__back.TT AND (#Z283_backward.T > T#5S);   // Z283_zur
      (C)     N    "GraDB_SK".noAction
   END_STEP
   TRANSITION Z283__back FROM Z283_backward TO Z284_backward   // T43
      := "AlwaysFALSE";
   END_TRANSITION
   STEP Z284_backward:   // S44, max time T#10S, warning time T#7S: Step commentary / Schrittkommentar
      interlock C := "AlwaysFALSE";   // Z284_zur
      supervision V := NOT #Z284__back.TT AND (#Z284_backward.T > T#5S);   // Z284_zur
      (C)     N    "GraDB_SK".noAction
   END_STEP
   TRANSITION Z284__back FROM Z284_backward TO Z285_backward   // T44
      := "AlwaysFALSE";
   END_TRANSITION
   STEP Z285_backward:   // S45, max time T#10S, warning time T#7S: Step commentary / Schrittkommentar
      interlock C := "AlwaysFALSE";   // Z285_zur
      supervision V := NOT #Z285__back.TT AND (#Z285_backward.T > T#5S);   // Z285_zur
      (C)     N    "GraDB_SK".noAction
   END_STEP
   TRANSITION Z285__back FROM Z285_backward TO Z286_backward   // T45
      := "AlwaysFALSE";
   END_TRANSITION
   STEP Z281_forward:   // S141, max time T#10S, warning time T#7S
      interlock C := "AlwaysFALSE";   // Z281_vor
      supervision V := NOT #Z281_in_front.TT AND (#Z281_forward.T > T#5S);   // Z281_vor
      (C)     N    "GraDB_SK".noAction
   END_STEP
   TRANSITION Z281_in_front FROM Z281_forward TO Z282_forward   // T141
      := "AlwaysFALSE";
   END_TRANSITION
   STEP Z282_forward:   // S142, max time T#10S, warning time T#7S
      interlock C := "AlwaysFALSE";   // Z282_vor
      supervision V := NOT #Z282_in_front.TT AND (#Z282_forward.T > T#5S);   // Z282_vor
      (C)     N    "GraDB_SK".noAction
   END_STEP
   TRANSITION Z282_in_front FROM Z282_forward TO Z283_forward   // T142
      := "AlwaysFALSE";
   END_TRANSITION
   STEP Z283_forward:   // S143, max time T#10S, warning time T#7S
      interlock C := "AlwaysFALSE";   // Z283_vor
      supervision V := NOT #Z283_in_front.TT AND (#Z283_forward.T > T#5S);   // Z283_vor
      (C)     N    "GraDB_SK".noAction
   END_STEP
   TRANSITION Z283_in_front FROM Z283_forward TO Z284_forward   // T143
      := "AlwaysFALSE";
   END_TRANSITION
   STEP Z284_forward:   // S144, max time T#10S, warning time T#7S
      interlock C := "AlwaysFALSE";   // Z284_vor
      supervision V := NOT #Z284_in_front.TT AND (#Z284_forward.T > T#5S);   // Z284_vor
      (C)     N    "GraDB_SK".noAction
   END_STEP
   TRANSITION Z284_in_front FROM Z284_forward TO Z285_forward   // T144
      := "AlwaysFALSE";
   END_TRANSITION
   STEP Z285_forward:   // S145, max time T#10S, warning time T#7S
      interlock C := "AlwaysFALSE";   // Z285_vor
      supervision V := NOT #Z285_in_front.TT AND (#Z285_forward.T > T#5S);   // Z285_vor
      (C)     N    "GraDB_SK".noAction
   END_STEP
   TRANSITION Z285_in_front FROM Z285_forward TO Z286_forward   // T145
      := "AlwaysFALSE";
   END_TRANSITION
   STEP Z286_backward:   // S46, max time T#10S, warning time T#7S: Step commentary / Schrittkommentar
      interlock C := "AlwaysFALSE";   // Z286_zur
      supervision V := NOT #Z286__back.TT AND (#Z286_backward.T > T#5S);   // Z286_zur
      (C)     N    "GraDB_SK".noAction
   END_STEP
   TRANSITION Z286__back FROM Z286_backward TO Z287_backward   // T46
      := "AlwaysFALSE";
   END_TRANSITION
   STEP Z287_backward:   // S47, max time T#10S, warning time T#7S: Step commentary / Schrittkommentar
      interlock C := "AlwaysFALSE";   // Z287_zur
      supervision V := NOT #Z287__back.TT AND (#Z287_backward.T > T#5S);   // Z287_zur
      (C)     N    "GraDB_SK".noAction
   END_STEP
   TRANSITION Z287__back FROM Z287_backward TO Z288_backward   // T47
      := "AlwaysFALSE";
   END_TRANSITION
   STEP Z288_backward:   // S48, max time T#10S, warning time T#7S: Step commentary / Schrittkommentar
      interlock C := "AlwaysFALSE";   // Z288_zur
      supervision V := NOT #Z288__back.TT AND (#Z288_backward.T > T#5S);   // Z288_zur
      (C)     N    "GraDB_SK".noAction
   END_STEP
   TRANSITION Z288__back FROM Z288_backward TO Z289_backward   // T48
      := "AlwaysFALSE";
   END_TRANSITION
   STEP Z289_backward:   // S49, max time T#10S, warning time T#7S: Step commentary / Schrittkommentar
      interlock C := "AlwaysFALSE";   // Z289_zur
      supervision V := NOT #Z289__back.TT AND (#Z289_backward.T > T#5S);   // Z289_zur
      (C)     N    "GraDB_SK".noAction
   END_STEP
   TRANSITION Z289__back FROM Z289_backward TO Z290_backward   // T49
      := "AlwaysFALSE";
   END_TRANSITION
   STEP Z290_backward:   // S50, max time T#10S, warning time T#7S: Step commentary / Schrittkommentar
      interlock C := "AlwaysFALSE";   // Z290_zur
      supervision V := NOT #Z290__back.TT AND (#Z290_backward.T > T#5S);   // Z290_zur
      (C)     N    "GraDB_SK".noAction
   END_STEP
   TRANSITION Z290__back FROM Z290_backward TO Z291_backward   // T50
      := "AlwaysFALSE";
   END_TRANSITION
   STEP Z286_forward:   // S146, max time T#10S, warning time T#7S: Step commentary / Schrittkommentar
      interlock C := "AlwaysFALSE";   // Z286_vor
      supervision V := NOT #Z286_in_front.TT AND (#Z286_forward.T > T#5S);   // Z286_vor
      (C)     N    "GraDB_SK".noAction
   END_STEP
   TRANSITION Z286_in_front FROM Z286_forward TO Z287_forward   // T146
      := "AlwaysFALSE";
   END_TRANSITION
   STEP Z287_forward:   // S147, max time T#10S, warning time T#7S: Step commentary / Schrittkommentar
      interlock C := "AlwaysFALSE";   // Z287_vor
      supervision V := NOT #Z287_in_front.TT AND (#Z287_forward.T > T#5S);   // Z287_vor
      (C)     N    "GraDB_SK".noAction
   END_STEP
   TRANSITION Z287_in_front FROM Z287_forward TO Z288_forward   // T147
      := "AlwaysFALSE";
   END_TRANSITION
   STEP Z288_forward:   // S148, max time T#10S, warning time T#7S: Step commentary / Schrittkommentar
      interlock C := "AlwaysFALSE";   // Z288_vor
      supervision V := NOT #Z288_in_front.TT AND (#Z288_forward.T > T#5S);   // Z288_vor
      (C)     N    "GraDB_SK".noAction
   END_STEP
   TRANSITION Z288_in_front FROM Z288_forward TO Z289_forward   // T148
      := "AlwaysFALSE";
   END_TRANSITION
   STEP Z289_forward:   // S149, max time T#10S, warning time T#7S: Step commentary / Schrittkommentar
      interlock C := "AlwaysFALSE";   // Z289_vor
      supervision V := NOT #Z289_in_front.TT AND (#Z289_forward.T > T#5S);   // Z289_vor
      (C)     N    "GraDB_SK".noAction
   END_STEP
   TRANSITION Z289_in_front FROM Z289_forward TO Z290_forward   // T149
      := "AlwaysFALSE";
   END_TRANSITION
   STEP Z290_forward:   // S150, max time T#10S, warning time T#7S: Step commentary / Schrittkommentar
      interlock C := "AlwaysFALSE";   // Z290_vor
      supervision V := NOT #Z290_in_front.TT AND (#Z290_forward.T > T#5S);   // Z290_vor
      (C)     N    "GraDB_SK".noAction
   END_STEP
   TRANSITION Z290_in_front FROM Z290_forward TO Z291_forward   // T150
      := "AlwaysFALSE";
   END_TRANSITION
   STEP Z291_backward:   // S51, max time T#10S, warning time T#7S: Step commentary / Schrittkommentar
      interlock C := "AlwaysFALSE";   // Z291_zur
      supervision V := NOT #Z291__back.TT AND (#Z291_backward.T > T#5S);   // Z291_zur
      (C)     N    "GraDB_SK".noAction
   END_STEP
   TRANSITION Z291__back FROM Z291_backward TO Z292_backward   // T51
      := "AlwaysFALSE";
   END_TRANSITION
   STEP Z292_backward:   // S52, max time T#10S, warning time T#7S: Step commentary / Schrittkommentar
      interlock C := "AlwaysFALSE";   // Z292_zur
      supervision V := NOT #Z292__back.TT AND (#Z292_backward.T > T#5S);   // Z292_zur
      (C)     N    "GraDB_SK".noAction
   END_STEP
   TRANSITION Z292__back FROM Z292_backward TO Z293_backward   // T52
      := "AlwaysFALSE";
   END_TRANSITION
   STEP Z293_backward:   // S53, max time T#10S, warning time T#7S: Step commentary / Schrittkommentar
      interlock C := "AlwaysFALSE";   // Z293_zur
      supervision V := NOT #Z293__back.TT AND (#Z293_backward.T > T#5S);   // Z293_zur
      (C)     N    "GraDB_SK".noAction
   END_STEP
   TRANSITION Z293__back FROM Z293_backward TO Z294_backward   // T53
      := "AlwaysFALSE";
   END_TRANSITION
   STEP Z294_backward:   // S54, max time T#10S, warning time T#7S: Step commentary / Schrittkommentar
      interlock C := "AlwaysFALSE";   // Z294_zur
      supervision V := NOT #Z294__back.TT AND (#Z294_backward.T > T#5S);   // Z294_zur
      (C)     N    "GraDB_SK".noAction
   END_STEP
   TRANSITION Z294__back FROM Z294_backward TO Z295_backward   // T54
      := "AlwaysFALSE";
   END_TRANSITION
   STEP Z295_backward:   // S55, max time T#10S, warning time T#7S: Step commentary / Schrittkommentar
      interlock C := "AlwaysFALSE";   // Z295_zur
      supervision V := NOT #Z295__back.TT AND (#Z295_backward.T > T#5S);   // Z295_zur
      (C)     N    "GraDB_SK".noAction
   END_STEP
   TRANSITION Z295__back FROM Z295_backward TO Z296_backward   // T55
      := "AlwaysFALSE";
   END_TRANSITION
   STEP Z296_backward:   // S56, max time T#10S, warning time T#7S: Step commentary / Schrittkommentar
      interlock C := "AlwaysFALSE";   // Z296_zur
      supervision V := NOT #Z296__back.TT AND (#Z296_backward.T > T#5S);   // Z296_zur
      (C)     N    "GraDB_SK".noAction
   END_STEP
   TRANSITION Z296__back FROM Z296_backward TO Z297_backward   // T56
      := "AlwaysFALSE";
   END_TRANSITION
   STEP Z297_backward:   // S57, max time T#10S, warning time T#7S: Step commentary / Schrittkommentar
      interlock C := "AlwaysFALSE";   // Z297_zur
      supervision V := NOT #Z297__back.TT AND (#Z297_backward.T > T#5S);   // Z297_zur
      (C)     N    "GraDB_SK".noAction
   END_STEP
   TRANSITION Z297__back FROM Z297_backward TO Z298_backward   // T57
      := "AlwaysFALSE";
   END_TRANSITION
   STEP Z298_backward:   // S58, max time T#10S, warning time T#7S: Step commentary / Schrittkommentar
      interlock C := "AlwaysFALSE";   // Z298_zur
      supervision V := NOT #Z298__back.TT AND (#Z298_backward.T > T#5S);   // Z298_zur
      (C)     N    "GraDB_SK".noAction
   END_STEP
   TRANSITION Z298__back FROM Z298_backward TO Z299_backward   // T58
      := "AlwaysFALSE";
   END_TRANSITION
   STEP Z299_backward:   // S59, max time T#10S, warning time T#7S: Step commentary / Schrittkommentar
      interlock C := "AlwaysFALSE";   // Z299_zur
      supervision V := NOT #Z299__back.TT AND (#Z299_backward.T > T#5S);   // Z299_zur
      (C)     N    "GraDB_SK".noAction
   END_STEP
   TRANSITION Z299__back FROM Z299_backward TO Z300_backward   // T59
      := "AlwaysFALSE";
   END_TRANSITION
   STEP Z300_backward:   // S60, max time T#10S, warning time T#7S: Step commentary / Schrittkommentar
      interlock C := "AlwaysFALSE";   // Z300_zur
      supervision V := NOT #Z300__back.TT AND (#Z300_backward.T > T#5S);   // Z300_zur
      (C)     N    "GraDB_SK".noAction
   END_STEP
   TRANSITION Z300__back FROM Z300_backward TO END   // T60
      := "AlwaysFALSE";
   END_TRANSITION
   STEP Z291_forward:   // S151, max time T#10S, warning time T#7S
      interlock C := "AlwaysFALSE";   // Z291_vor
      supervision V := NOT #Z291_in_front.TT AND (#Z291_forward.T > T#5S);   // Z291_vor
      (C)     N    "GraDB_SK".noAction
   END_STEP
   TRANSITION Z291_in_front FROM Z291_forward TO Z292_forward   // T151
      := "AlwaysFALSE";
   END_TRANSITION
   STEP Z292_forward:   // S152, max time T#10S, warning time T#7S
      interlock C := "AlwaysFALSE";   // Z292_vor
      supervision V := NOT #Z292_in_front.TT AND (#Z292_forward.T > T#5S);   // Z292_vor
      (C)     N    "GraDB_SK".noAction
   END_STEP
   TRANSITION Z292_in_front FROM Z292_forward TO Z293_forward   // T152
      := "AlwaysFALSE";
   END_TRANSITION
   STEP Z293_forward:   // S153, max time T#10S, warning time T#7S
      interlock C := "AlwaysFALSE";   // Z293_vor
      supervision V := NOT #Z293_in_front.TT AND (#Z293_forward.T > T#5S);   // Z293_vor
      (C)     N    "GraDB_SK".noAction
   END_STEP
   TRANSITION Z293_in_front FROM Z293_forward TO Z294_forward   // T153
      := "AlwaysFALSE";
   END_TRANSITION
   STEP Z294_forward:   // S154, max time T#10S, warning time T#7S
      interlock C := "AlwaysFALSE";   // Z294_vor
      supervision V := NOT #Z294_in_front.TT AND (#Z294_forward.T > T#5S);   // Z294_vor
      (C)     N    "GraDB_SK".noAction
   END_STEP
   TRANSITION Z294_in_front FROM Z294_forward TO Z295_forward   // T154
      := "AlwaysFALSE";
   END_TRANSITION
   STEP Z295_forward:   // S155, max time T#10S, warning time T#7S
      interlock C := "AlwaysFALSE";   // Z295_vor
      supervision V := NOT #Z295_in_front.TT AND (#Z295_forward.T > T#5S);   // Z295_vor
      (C)     N    "GraDB_SK".noAction
   END_STEP
   TRANSITION Z295_in_front FROM Z295_forward TO Z296_forward   // T155
      := "AlwaysFALSE";
   END_TRANSITION
   STEP Z296_forward:   // S156, max time T#10S, warning time T#7S: Step commentary / Schrittkommentar
      interlock C := "AlwaysFALSE";   // Z296_vor
      supervision V := NOT #Z296_in_front.TT AND (#Z296_forward.T > T#5S);   // Z296_vor
      (C)     N    "GraDB_SK".noAction
   END_STEP
   TRANSITION Z296_in_front FROM Z296_forward TO Z297_forward   // T156
      := "AlwaysFALSE";
   END_TRANSITION
   STEP Z297_forward:   // S157, max time T#10S, warning time T#7S: Step commentary / Schrittkommentar
      interlock C := "AlwaysFALSE";   // Z297_vor
      supervision V := NOT #Z297_in_front.TT AND (#Z297_forward.T > T#5S);   // Z297_vor
      (C)     N    "GraDB_SK".noAction
   END_STEP
   TRANSITION Z297_in_front FROM Z297_forward TO Z298_forward   // T157
      := "AlwaysFALSE";
   END_TRANSITION
   STEP Z298_forward:   // S158, max time T#10S, warning time T#7S: Step commentary / Schrittkommentar
      interlock C := "AlwaysFALSE";   // Z298_vor
      supervision V := NOT #Z298_in_front.TT AND (#Z298_forward.T > T#5S);   // Z298_vor
      (C)     N    "GraDB_SK".noAction
   END_STEP
   TRANSITION Z298_in_front FROM Z298_forward TO Z299_forward   // T158
      := "AlwaysFALSE";
   END_TRANSITION
   STEP Z299_forward:   // S159, max time T#10S, warning time T#7S: Step commentary / Schrittkommentar
      interlock C := "AlwaysFALSE";   // Z299_vor
      supervision V := NOT #Z299_in_front.TT AND (#Z299_forward.T > T#5S);   // Z299_vor
      (C)     N    "GraDB_SK".noAction
   END_STEP
   TRANSITION Z299_in_front FROM Z299_forward TO Z300_forward   // T159
      := "AlwaysFALSE";
   END_TRANSITION
   STEP Z300_forward:   // S160, max time T#10S, warning time T#7S: Step commentary / Schrittkommentar
      interlock C := "AlwaysFALSE";   // Z300_vor
      supervision V := NOT #Z300_in_front.TT AND (#Z300_forward.T > T#5S);   // Z300_vor
      (C)     N    "GraDB_SK".noAction
   END_STEP
   TRANSITION Z300_in_front FROM Z300_forward TO END   // T160
      := "AlwaysFALSE";
   END_TRANSITION

   // permanent post-instructions
   NETWORK 1
   TITLE = HMI Lite Pass on data / HMI Lite Daten weiterreichen
      "LTLL_ManualGraphInterlock"(ManualGraphExtOutput := #extBlock.output,
                              ManualGraphControlScreen := "LTLL_ManualGraphControl_OP70".screen[0]);
   NETWORK 2
   TITLE = Report step error / Schrittkettenfehler melden
      "SysFC_NumOfSQErrors"(FLT := #RT_DATA.SQ_FLAGS.ERR_FLT,
                            Fault_SQ := "AnwDB_OperatingModes_OP70".BA[0].error_report_SK,
                            NumOf_Fault_SQ := "AnwDB_ZP_Alarm_OP70".FaultsNoSK_ST1);
END_FUNCTION_BLOCK
